INTERFACE I_SimpleLogSource EXTENDS I_Base

{attribute 'monitoring':='call'}
PROPERTY SourceName : T_MaxString
GET
END_GET
END_PROPERTY

{attribute 'monitoring':='call'}
PROPERTY TimeStamp : T_FILETIME64
GET
END_GET
END_PROPERTY

END_INTERFACE

(* stored: Version 1.1.0.1
   Itf I_SimpleLogSource: Id {a5a2a655-616d-42a7-94d2-e761e8fdbc3b}
   Property SourceName: Id {dabf4b24-2b1e-4f8d-a1be-713080e33fc5}
   Get Get: Id {9a84ccc9-66ef-46b6-8b18-728c37609ee9}
   Property TimeStamp: Id {24d5e1ad-9cf4-44b2-a847-8639250614f6}
   Get Get: Id {427482e7-e897-4de6-b03e-8b2b7a04d550} *)
